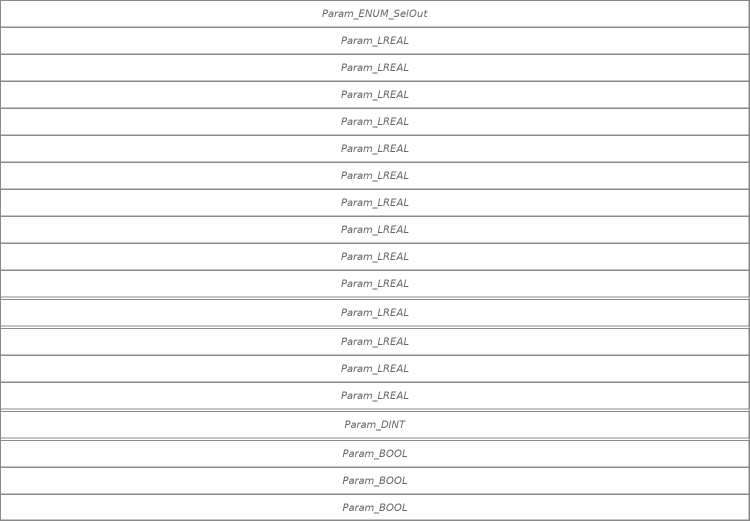
VISUALIZATION Visu_Mparam_Heat  // 750x521
    Frame (0,27 750x27)
        shows Param_LREAL(nIdx := 5)
    Frame (0,54 750x27)
        shows Param_LREAL(nIdx := 7)
    Frame (0,81 750x27)
        shows Param_LREAL(nIdx := 9)
    Frame (0,108 750x27)
        shows Param_LREAL(nIdx := 11)
    Frame (0,411 750x27)
        shows Param_DINT(nIdx := 10)
    Frame (0,0 750x27)
        shows Param_ENUM_SelOut(nIdx := 2)
    Frame (0,135 750x27)
        shows Param_LREAL(nIdx := 12)
    Frame (0,162 750x27)
        shows Param_LREAL(nIdx := 13)
    Frame (0,189 750x27)
        shows Param_LREAL(nIdx := 14)
    Frame (0,216 750x27)
        shows Param_LREAL(nIdx := 15)
    Frame (0,243 750x27)
        shows Param_LREAL(nIdx := 17)
    Frame (0,270 750x27)
        shows Param_LREAL(nIdx := 18)
    Frame (0,299 750x27)
        shows Param_LREAL(nIdx := 22)
    Frame (0,328 750x27)
        shows Param_LREAL(nIdx := 33)
    Frame (0,355 750x27)
        shows Param_LREAL(nIdx := 34)
    Frame (0,382 750x27)
        shows Param_LREAL(nIdx := 36)
    Frame (0,440 750x27)
        shows Param_BOOL(nIdx := 12)
    Frame (0,467 750x27)
        shows Param_BOOL(nIdx := 16)
    Frame (0,494 750x27)
        shows Param_BOOL(nIdx := 19)
END_VISUALIZATION

(* stored: Version 1.1.0.1
   Visu Visu_Mparam_Heat: Id {dd7220ea-a780-43a3-ab41-0e9437711069} *)
